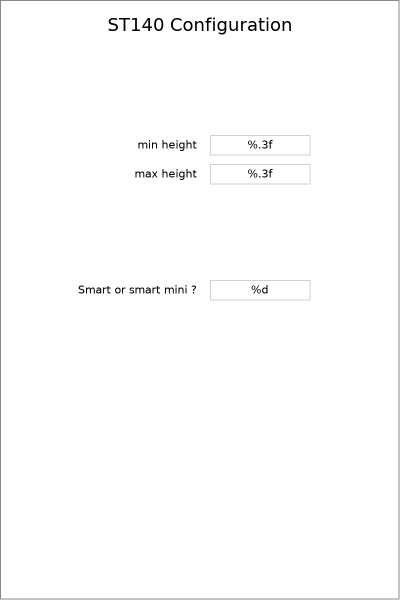
VISUALIZATION VISU_Recipe_ST140  // 400x600
    Label (0,5 400x40), "ST140 Configuration"
    Label (0,280 200x20), "Smart or smart mini ?"
    Textfield (210,280 100x20), "%d", text variable: _20_AUTO.recipe.st140.xIsTypeMiniOrSmart
        OnMouseDown: write the text variable via Default
    Label (0,135 200x20), "min height"
    Textfield (210,135 100x20), "%.3f", text variable: _20_AUTO.recipe.st140.rMinHeightSensor
        OnMouseDown: write the text variable via Default
    Label (0,164 200x20), "max height"
    Textfield (210,164 100x20), "%.3f", text variable: _20_AUTO.recipe.st140.rMaxHeightSensor
        OnMouseDown: write the text variable via Default
END_VISUALIZATION

(* stored: Version 1.1.0.1, ProductVersion 3.1.4024.6
   Visu VISU_Recipe_ST140: Id {2e95b056-fb3c-479d-8cb3-075dee377010} *)
